(* IEC 61131-3 sources: Fisk_Test/Fisk.fbsproj/MyController.device.xml.v3^/Plc Logic.plclogic.xml.v3^/Application.application.xml.v3^, 6 files *)

(* ---- GVL.gvl ---- *)
{attribute 'qualified_only'}
VAR_GLOBAL
    myVar:BOOL;
END_VAR

(* ---- EM01.prg.st ---- *)
PROGRAM EM01
VAR
	Counter: INT;
END_VAR

Counter := Counter +1;

(* ---- EM02.prg.st ---- *)
PROGRAM EM02
VAR
END_VAR

(* ---- MAST.prg.st ---- *)
PROGRAM MAST
VAR
END_VAR

(* ---- Merge.prg.st ---- *)
PROGRAM Merge
VAR
	Counter: INT;
END_VAR

Counter := Counter + 2 ;

(* ---- SR_Main.prg.st ---- *)
PROGRAM SR_Main
VAR
	Counter: INT;
END_VAR

Counter := Counter + 2 ;
